// TwinCAT 3 PLC project Motion_TST
// ProgramVersion: 3.1.4022.7
// libraries:
//   lcls-twincat-motion, * (SLAC)
//   Tc2_Standard, * (Beckhoff Automation GmbH)
//   Tc2_System, * (Beckhoff Automation GmbH)
//   Tc3_Module, * (Beckhoff Automation GmbH)
// project tree:
//   / PlcTask.TcTTO
//   POUs/ MAIN.TcPOU
// real-time tasks:
//   TASK PlcTask: cycle T#10ms, priority 20, ADS port 350
// motion (NC):
// I/O:
//   DEVICE Device 1 (EtherCAT)
// variable links:
//   Motion_TST Instance <-> Device 1 (EtherCAT)/Term 1 (EK1200)/Term 3 (EL1084)
//     PlcTask Inputs/MAIN.bLimitBackwardEnable <-> Channel 1/Input
//     PlcTask Inputs/MAIN.bLimitForwardEnable <-> Channel 2/Input
//   Motion_TST Instance <-> Device 1 (EtherCAT)/Term 1 (EK1200)/Term 4 (EL5042)
//     PlcTask Inputs/MAIN.M1.nRawEncoderULINT <-> FB Inputs Channel 1/Position
//   Motion_TST Instance <-> NC-Task 1 SAF/Axes/Axis 1
//     PlcTask Inputs/MAIN.M1.Axis.NcToPlc <-> Outputs/ToPlc
//     PlcTask Outputs/MAIN.M1.Axis.PlcToNc <-> Inputs/FromPlc

CONFIGURATION Motion_TST
    RESOURCE PLC ON TwinCAT3
        TASK PlcTask(INTERVAL := T#10ms, PRIORITY := 20);
        PROGRAM MAIN WITH PlcTask : MAIN;
    END_RESOURCE
END_CONFIGURATION

// ---- POUs/MAIN.TcPOU
PROGRAM MAIN
VAR
	// Define EPICS interface (struct) for moving motor
	{attribute 'pytmc' := 'pv: PRACTICE:PLC_MOT'}
	{attribute 'TcLinkTo' := '.nRawEncoderULINT     := TIID^Device 1 (EtherCAT)^Term 1 (EK1200)^Term 4 (EL5042)^FB Inputs Channel 1^Position'}
	M1: ST_MotionStage := (sName := 'PRACTICE:PLC_MOT',
                        bPowerSelf := TRUE); // opt out of PMPS and handle motor enabling within FB_MotionStage

	// Attribute Linking Hardware
	// Inputs (limit switch)
	{attribute 'TcLinkTo' := 'TIID^Device 1 (EtherCAT)^Term 1 (EK1200)^Term 3 (EL1084)^Channel 1^Input'}
	bLimitBackwardEnable AT %I* : BOOL;

	{attribute 'TcLinkTo' := 'TIID^Device 1 (EtherCAT)^Term 1 (EK1200)^Term 3 (EL1084)^Channel 2^Input'}
	bLimitForwardEnable AT %I* : BOOL;

	// Function Block logic
	fbMotion1 : FB_MotionStage;
END_VAR

// Limit switch is NPN, while motion library is uses PNP
M1.bLimitBackwardEnable := NOT bLimitBackwardEnable;
M1.bLimitForwardEnable := NOT bLimitForwardEnable;

M1.bHardwareEnable := TRUE; // ok to move

// Invoke function block call
fbMotion1(stMotionStage := M1);

END_PROGRAM
